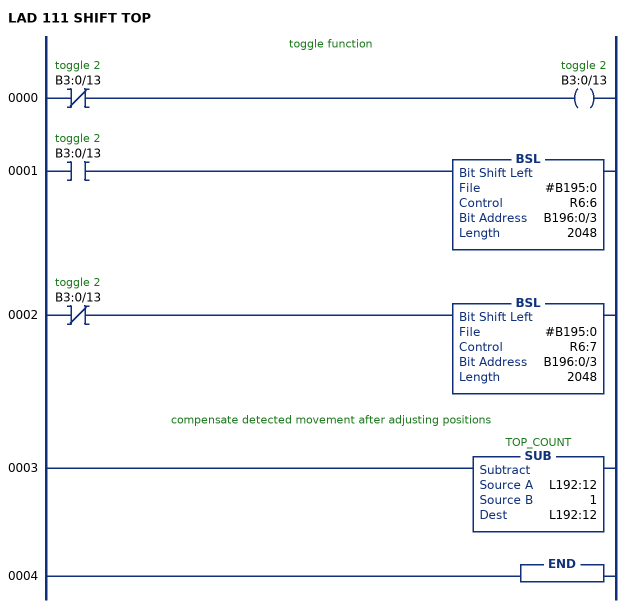
% Rung: 0 %
% toggle function %
SOR XIO B3:0/13 OTE B3:0/13 EOR
%   B3:0/13  "toggle 2" %
% Rung: 1 %
SOR XIC B3:0/13 BSL #B195:0 R6:6 B196:0/3 2048 EOR
%   B3:0/13  "toggle 2" %
%   B196:0/3  OFF %
% Rung: 2 %
SOR XIO B3:0/13 BSL #B195:0 R6:7 B196:0/3 2048 EOR
%   B3:0/13  "toggle 2" %
%   B196:0/3  OFF %
% Rung: 3 %
% compensate detected movement after adjusting positions %
SOR SUB L192:12 1 L192:12 EOR
%   L192:12  TOP_COUNT %
% Rung: 4 %
SOR END EOR

LADDER 121 "OPTIC BOT"
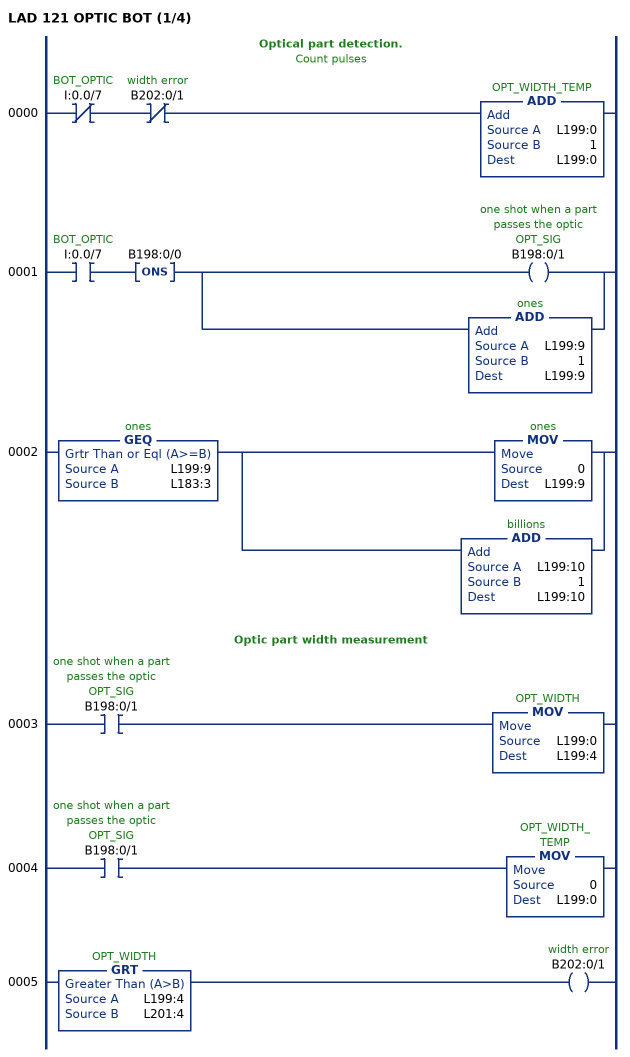
% Rung: 0 %
% TITLE: Optical part detection. %
% Count pulses %
SOR XIO I:0.0/7 XIO B202:0/1 ADD L199:0 1 L199:0 EOR
%   I:0.0/7  BOT_OPTIC %
%   B202:0/1  "width error" %
%   L199:0  OPT_WIDTH_TEMP %
% Rung: 1 %
SOR XIC I:0.0/7 ONS B198:0/0 BST OTE B198:0/1 NXB ADD L199:9 1 L199:9 BND EOR
%   I:0.0/7  BOT_OPTIC %
%   B198:0/1  OPT_SIG  "one shot when a part passes the optic" %
%   L199:9  "ones" %
% Rung: 2 %
SOR GEQ L199:9 L183:3 BST MOV 0 L199:9 NXB ADD L199:10 1 L199:10 BND EOR
%   L199:9  "ones" %
%   L183:3  "button state" %
%   L199:10  "billions" %
% Rung: 3 %
% TITLE: Optic part width measurement %
SOR XIC B198:0/1 MOV L199:0 L199:4 EOR
%   B198:0/1  OPT_SIG  "one shot when a part passes the optic" %
%   L199:0  OPT_WIDTH_TEMP %
%   L199:4  OPT_WIDTH %
% Rung: 4 %
SOR XIC B198:0/1 MOV 0 L199:0 EOR
%   B198:0/1  OPT_SIG  "one shot when a part passes the optic" %
%   L199:0  OPT_WIDTH_TEMP %
% Rung: 5 %
SOR GRT L199:4 L201:4 OTE B202:0/1 EOR
%   L199:4  OPT_WIDTH %
%   L201:4  MAX_WIDTH  "hmi in" %
%   B202:0/1  "width error" %

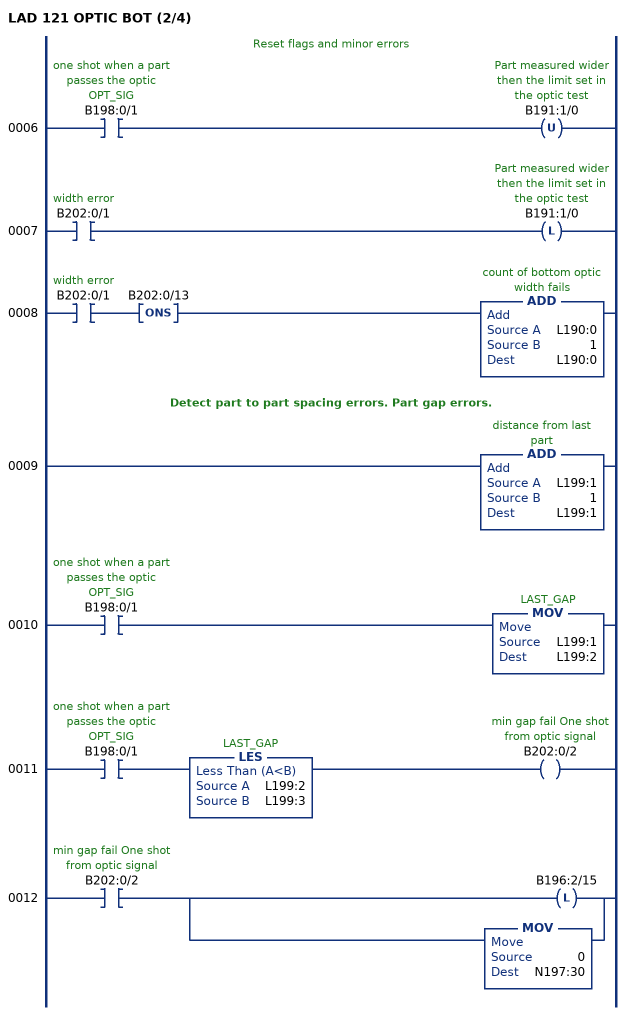
% Rung: 6 %
% Reset flags and minor errors %
SOR XIC B198:0/1 OTU B191:1/0 EOR
%   B198:0/1  OPT_SIG  "one shot when a part passes the optic" %
%   B191:1/0  "Part measured wider then the limit set in the optic test" %
% Rung: 7 %
SOR XIC B202:0/1 OTL B191:1/0 EOR
%   B202:0/1  "width error" %
%   B191:1/0  "Part measured wider then the limit set in the optic test" %
% Rung: 8 %
SOR XIC B202:0/1 ONS B202:0/13 ADD L190:0 1 L190:0 EOR
%   B202:0/1  "width error" %
%   L190:0  "count of bottom optic width fails" %
% Rung: 9 %
% TITLE: Detect part to part spacing errors. Part gap errors. %
SOR ADD L199:1 1 L199:1 EOR
%   L199:1  "distance from last part" %
% Rung: 10 %
SOR XIC B198:0/1 MOV L199:1 L199:2 EOR
%   B198:0/1  OPT_SIG  "one shot when a part passes the optic" %
%   L199:1  "distance from last part" %
%   L199:2  LAST_GAP %
% Rung: 11 %
SOR XIC B198:0/1 LES L199:2 L199:3 OTE B202:0/2 EOR
%   B198:0/1  OPT_SIG  "one shot when a part passes the optic" %
%   L199:2  LAST_GAP %
%   L199:3  MIN_WIDTH %
%   B202:0/2  "min gap fail One shot from optic signal" %
% Rung: 12 %
SOR XIC B202:0/2 BST OTL B196:2/15 NXB MOV 0 N197:30 BND EOR
%   B202:0/2  "min gap fail One shot from optic signal" %

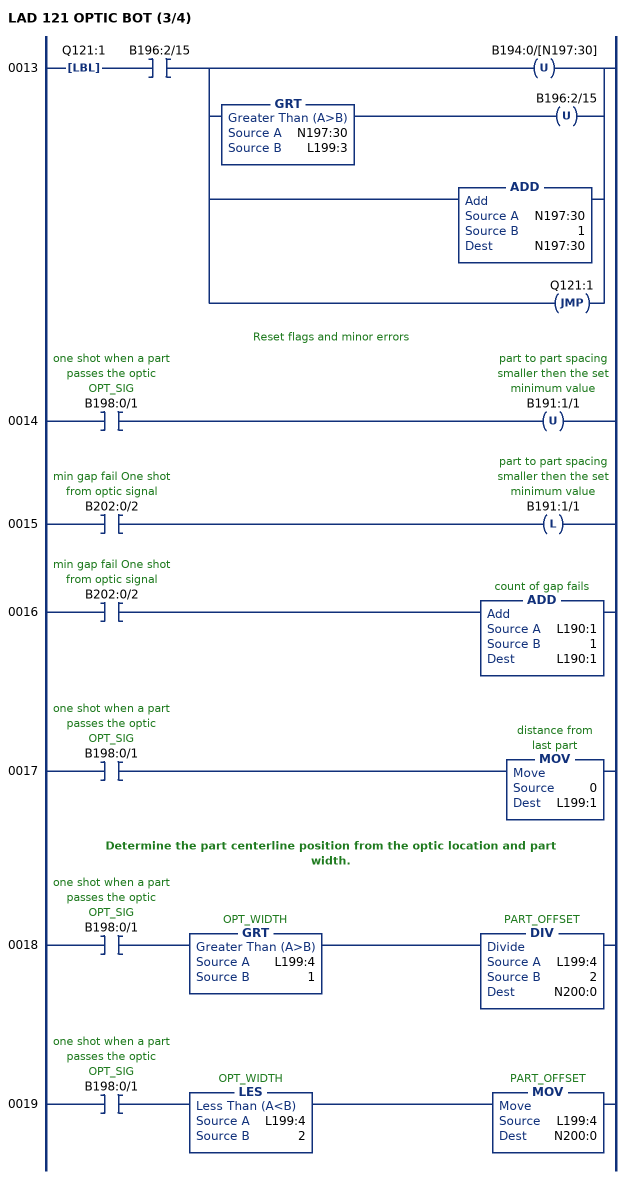
% Rung: 13 %
SOR LBL Q121:1 XIC B196:2/15 BST OTU B194:0/[N197:30] NXB GRT N197:30 L199:3 OTU B196:2/15 NXB ADD N197:30 1 N197:30 NXB JMP Q121:1 BND EOR
%   L199:3  MIN_WIDTH %
% Rung: 14 %
% Reset flags and minor errors %
SOR XIC B198:0/1 OTU B191:1/1 EOR
%   B198:0/1  OPT_SIG  "one shot when a part passes the optic" %
%   B191:1/1  "part to part spacing smaller then the set minimum value" %
% Rung: 15 %
SOR XIC B202:0/2 OTL B191:1/1 EOR
%   B202:0/2  "min gap fail One shot from optic signal" %
%   B191:1/1  "part to part spacing smaller then the set minimum value" %
% Rung: 16 %
SOR XIC B202:0/2 ADD L190:1 1 L190:1 EOR
%   B202:0/2  "min gap fail One shot from optic signal" %
%   L190:1  "count of gap fails" %
% Rung: 17 %
SOR XIC B198:0/1 MOV 0 L199:1 EOR
%   B198:0/1  OPT_SIG  "one shot when a part passes the optic" %
%   L199:1  "distance from last part" %
% Rung: 18 %
% TITLE: Determine the part centerline position from the optic location and part width. %
SOR XIC B198:0/1 GRT L199:4 1 DIV L199:4 2 N200:0 EOR
%   B198:0/1  OPT_SIG  "one shot when a part passes the optic" %
%   L199:4  OPT_WIDTH %
%   N200:0  PART_OFFSET %
% Rung: 19 %
SOR XIC B198:0/1 LES L199:4 2 MOV L199:4 N200:0 EOR
%   B198:0/1  OPT_SIG  "one shot when a part passes the optic" %
%   L199:4  OPT_WIDTH %
%   N200:0  PART_OFFSET %

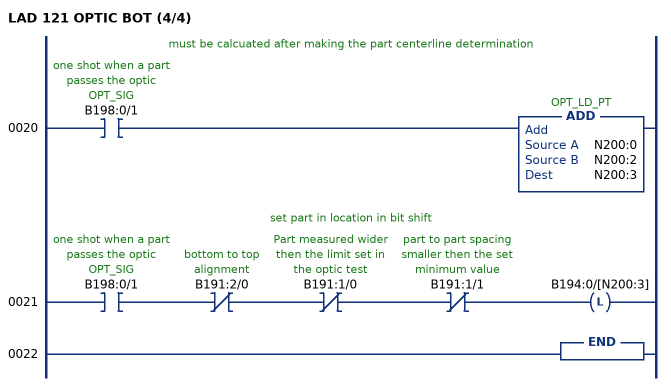
% Rung: 20 %
% must be calcuated after making the part centerline determination %
SOR XIC B198:0/1 ADD N200:0 N200:2 N200:3 EOR
%   B198:0/1  OPT_SIG  "one shot when a part passes the optic" %
%   N200:0  PART_OFFSET %
%   N200:2  OPTIC_LOC %
%   N200:3  OPT_LD_PT %
% Rung: 21 %
% set part in location in bit shift %
SOR XIC B198:0/1 XIO B191:2/0 XIO B191:1/0 XIO B191:1/1 OTL B194:0/[N200:3] EOR
%   B198:0/1  OPT_SIG  "one shot when a part passes the optic" %
%   B191:2/0  "bottom to top alignment" %
%   B191:1/0  "Part measured wider then the limit set in the optic test" %
%   B191:1/1  "part to part spacing smaller then the set minimum value" %
%   N200:3  OPT_LD_PT %
% Rung: 22 %
SOR END EOR

LADDER 125 "INS 1"
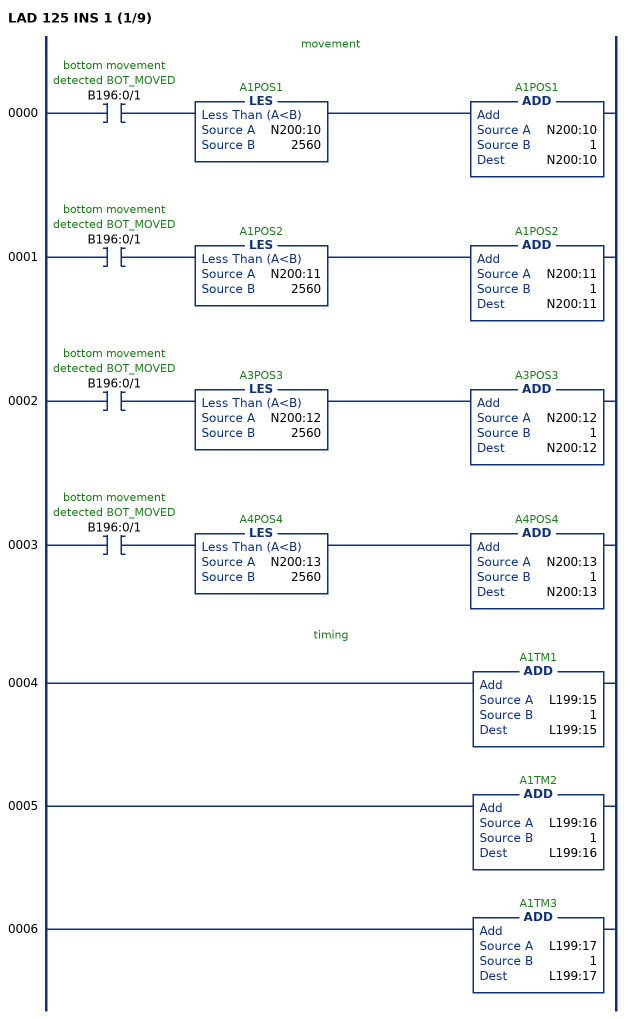
% Rung: 0 %
% movement %
SOR XIC B196:0/1 LES N200:10 2560 ADD N200:10 1 N200:10 EOR
%   B196:0/1  BOT_MOVED  "bottom movement detected" %
%   N200:10  A1POS1 %
% Rung: 1 %
SOR XIC B196:0/1 LES N200:11 2560 ADD N200:11 1 N200:11 EOR
%   B196:0/1  BOT_MOVED  "bottom movement detected" %
%   N200:11  A1POS2 %
% Rung: 2 %
SOR XIC B196:0/1 LES N200:12 2560 ADD N200:12 1 N200:12 EOR
%   B196:0/1  BOT_MOVED  "bottom movement detected" %
%   N200:12  A3POS3 %
% Rung: 3 %
SOR XIC B196:0/1 LES N200:13 2560 ADD N200:13 1 N200:13 EOR
%   B196:0/1  BOT_MOVED  "bottom movement detected" %
%   N200:13  A4POS4 %
% Rung: 4 %
% timing %
SOR ADD L199:15 1 L199:15 EOR
%   L199:15  A1TM1 %
% Rung: 5 %
SOR ADD L199:16 1 L199:16 EOR
%   L199:16  A1TM2 %
% Rung: 6 %
SOR ADD L199:17 1 L199:17 EOR
%   L199:17  A1TM3 %

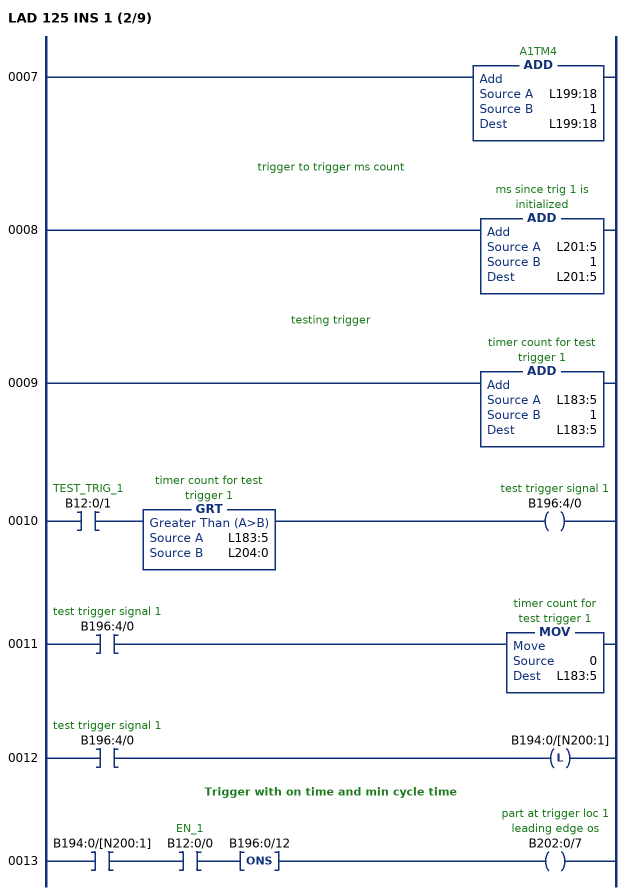
% Rung: 7 %
SOR ADD L199:18 1 L199:18 EOR
%   L199:18  A1TM4 %
% Rung: 8 %
% trigger to trigger ms count %
SOR ADD L201:5 1 L201:5 EOR
%   L201:5  "ms since trig 1 is initialized" %
% Rung: 9 %
% testing trigger %
SOR ADD L183:5 1 L183:5 EOR
%   L183:5  "timer count for test trigger 1" %
% Rung: 10 %
SOR XIC B12:0/1 GRT L183:5 L204:0 OTE B196:4/0 EOR
%   B12:0/1  TEST_TRIG_1 %
%   L183:5  "timer count for test trigger 1" %
%   B196:4/0  "test trigger signal 1" %
% Rung: 11 %
SOR XIC B196:4/0 MOV 0 L183:5 EOR
%   B196:4/0  "test trigger signal 1" %
%   L183:5  "timer count for test trigger 1" %
% Rung: 12 %
SOR XIC B196:4/0 OTL B194:0/[N200:1] EOR
%   B196:4/0  "test trigger signal 1" %
%   N200:1  INS_1_TRIG_LOC %
% Rung: 13 %
% TITLE: Trigger with on time and min cycle time %
SOR XIC B194:0/[N200:1] XIC B12:0/0 ONS B196:0/12 OTE B202:0/7 EOR
%   N200:1  INS_1_TRIG_LOC %
%   B12:0/0  EN_1 %
%   B202:0/7  "part at trigger loc 1 leading edge os" %

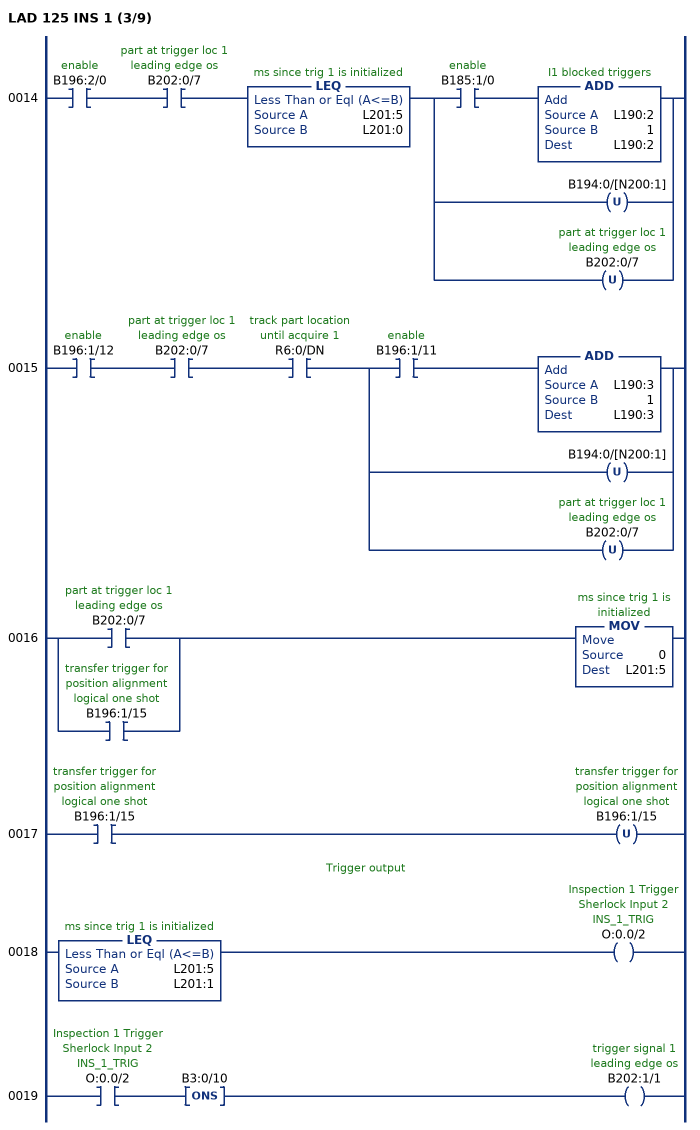
% Rung: 14 %
SOR XIC B196:2/0 XIC B202:0/7 LEQ L201:5 L201:0 BST XIC B185:1/0 ADD L190:2 1 L190:2 NXB OTU B194:0/[N200:1] NXB OTU B202:0/7 BND EOR
%   B196:2/0  "enable" %
%   B202:0/7  "part at trigger loc 1 leading edge os" %
%   L201:5  "ms since trig 1 is initialized" %
%   L201:0  CAM_1_MIN_CYCLE_TIME %
%   B185:1/0  "enable" %
%   L190:2  "I1 blocked triggers" %
%   N200:1  INS_1_TRIG_LOC %
% Rung: 15 %
SOR XIC B196:1/12 XIC B202:0/7 XIC R6:0/DN BST XIC B196:1/11 ADD L190:3 1 L190:3 NXB OTU B194:0/[N200:1] NXB OTU B202:0/7 BND EOR
%   B196:1/12  "enable" %
%   B202:0/7  "part at trigger loc 1 leading edge os" %
%   R6:0  "track part location until acquire 1" %
%   B196:1/11  "enable" %
%   N200:1  INS_1_TRIG_LOC %
% Rung: 16 %
SOR BST XIC B202:0/7 NXB XIC B196:1/15 BND MOV 0 L201:5 EOR
%   B202:0/7  "part at trigger loc 1 leading edge os" %
%   B196:1/15  "transfer trigger for position alignment logical one shot" %
%   L201:5  "ms since trig 1 is initialized" %
% Rung: 17 %
SOR XIC B196:1/15 OTU B196:1/15 EOR
%   B196:1/15  "transfer trigger for position alignment logical one shot" %
% Rung: 18 %
% Trigger output %
SOR LEQ L201:5 L201:1 OTE O:0.0/2 EOR
%   L201:5  "ms since trig 1 is initialized" %
%   L201:1  CAM_1_TRIG_TIME  "out time" %
%   O:0.0/2  INS_1_TRIG  "Inspection 1 Trigger Sherlock Input 2" %
% Rung: 19 %
SOR XIC O:0.0/2 ONS B3:0/10 OTE B202:1/1 EOR
%   O:0.0/2  INS_1_TRIG  "Inspection 1 Trigger Sherlock Input 2" %
%   B202:1/1  "trigger signal 1 leading edge os" %

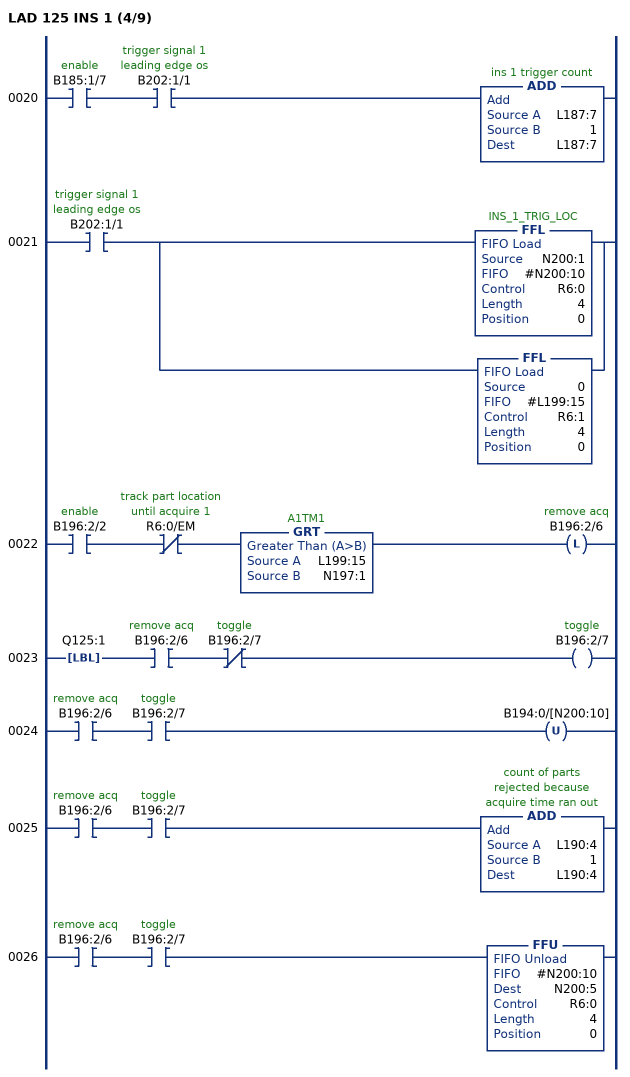
% Rung: 20 %
SOR XIC B185:1/7 XIC B202:1/1 ADD L187:7 1 L187:7 EOR
%   B185:1/7  "enable" %
%   B202:1/1  "trigger signal 1 leading edge os" %
%   L187:7  "ins 1 trigger count" %
% Rung: 21 %
SOR XIC B202:1/1 BST FFL N200:1 #N200:10 R6:0 4 0 NXB FFL 0 #L199:15 R6:1 4 0 BND EOR
%   B202:1/1  "trigger signal 1 leading edge os" %
%   N200:1  INS_1_TRIG_LOC %
%   N200:10  A1POS1 %
%   R6:0  "track part location until acquire 1" %
%   L199:15  A1TM1 %
%   R6:1  "track acquire time 1" %
% Rung: 22 %
SOR XIC B196:2/2 XIO R6:0/EM GRT L199:15 N197:1 OTL B196:2/6 EOR
%   B196:2/2  "enable" %
%   R6:0  "track part location until acquire 1" %
%   L199:15  A1TM1 %
%   N197:1  "maximim acquire time 1" %
%   B196:2/6  "remove acq" %
% Rung: 23 %
SOR LBL Q125:1 XIC B196:2/6 XIO B196:2/7 OTE B196:2/7 EOR
%   B196:2/6  "remove acq" %
%   B196:2/7  "toggle" %
% Rung: 24 %
SOR XIC B196:2/6 XIC B196:2/7 OTU B194:0/[N200:10] EOR
%   B196:2/6  "remove acq" %
%   B196:2/7  "toggle" %
%   N200:10  A1POS1 %
% Rung: 25 %
SOR XIC B196:2/6 XIC B196:2/7 ADD L190:4 1 L190:4 EOR
%   B196:2/6  "remove acq" %
%   B196:2/7  "toggle" %
%   L190:4  "count of parts rejected because acquire time ran out" %
% Rung: 26 %
SOR XIC B196:2/6 XIC B196:2/7 FFU #N200:10 N200:5 R6:0 4 0 EOR
%   B196:2/6  "remove acq" %
%   B196:2/7  "toggle" %
%   N200:10  A1POS1 %
%   R6:0  "track part location until acquire 1" %

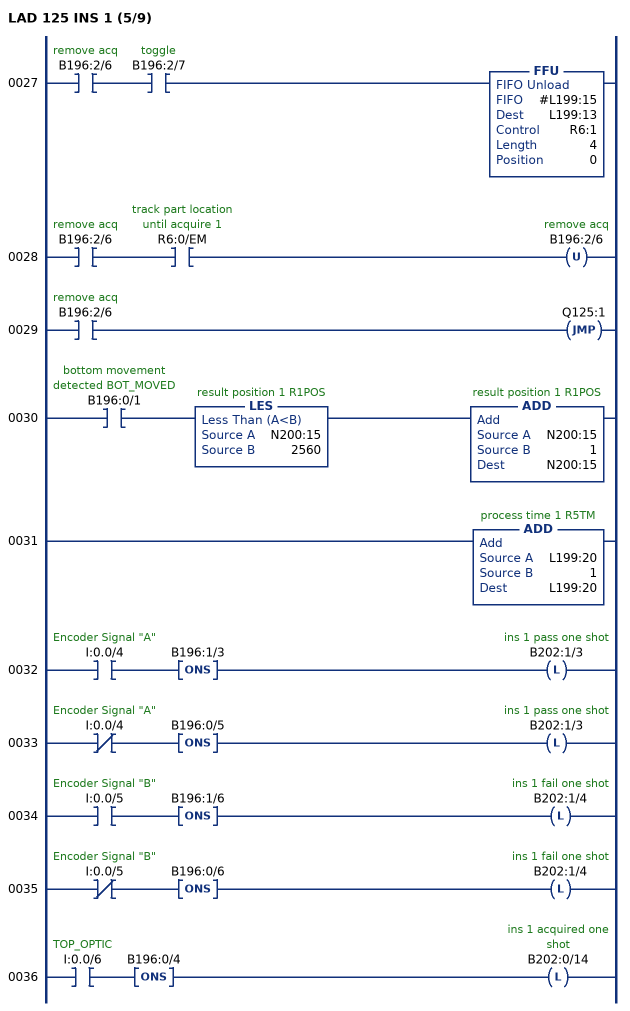
% Rung: 27 %
SOR XIC B196:2/6 XIC B196:2/7 FFU #L199:15 L199:13 R6:1 4 0 EOR
%   B196:2/6  "remove acq" %
%   B196:2/7  "toggle" %
%   L199:15  A1TM1 %
%   R6:1  "track acquire time 1" %
% Rung: 28 %
SOR XIC B196:2/6 XIC R6:0/EM OTU B196:2/6 EOR
%   B196:2/6  "remove acq" %
%   R6:0  "track part location until acquire 1" %
% Rung: 29 %
SOR XIC B196:2/6 JMP Q125:1 EOR
%   B196:2/6  "remove acq" %
% Rung: 30 %
SOR XIC B196:0/1 LES N200:15 2560 ADD N200:15 1 N200:15 EOR
%   B196:0/1  BOT_MOVED  "bottom movement detected" %
%   N200:15  R1POS  "result position 1" %
% Rung: 31 %
SOR ADD L199:20 1 L199:20 EOR
%   L199:20  R5TM  "process time 1" %
% Rung: 32 %
SOR XIC I:0.0/4 ONS B196:1/3 OTL B202:1/3 EOR
%   I:0.0/4  "Encoder Signal "A"" %
%   B202:1/3  "ins 1 pass one shot" %
% Rung: 33 %
SOR XIO I:0.0/4 ONS B196:0/5 OTL B202:1/3 EOR
%   I:0.0/4  "Encoder Signal "A"" %
%   B202:1/3  "ins 1 pass one shot" %
% Rung: 34 %
SOR XIC I:0.0/5 ONS B196:1/6 OTL B202:1/4 EOR
%   I:0.0/5  "Encoder Signal "B"" %
%   B202:1/4  "ins 1 fail one shot" %
% Rung: 35 %
SOR XIO I:0.0/5 ONS B196:0/6 OTL B202:1/4 EOR
%   I:0.0/5  "Encoder Signal "B"" %
%   B202:1/4  "ins 1 fail one shot" %
% Rung: 36 %
SOR XIC I:0.0/6 ONS B196:0/4 OTL B202:0/14 EOR
%   I:0.0/6  TOP_OPTIC %
%   B202:0/14  "ins 1 acquired one shot" %

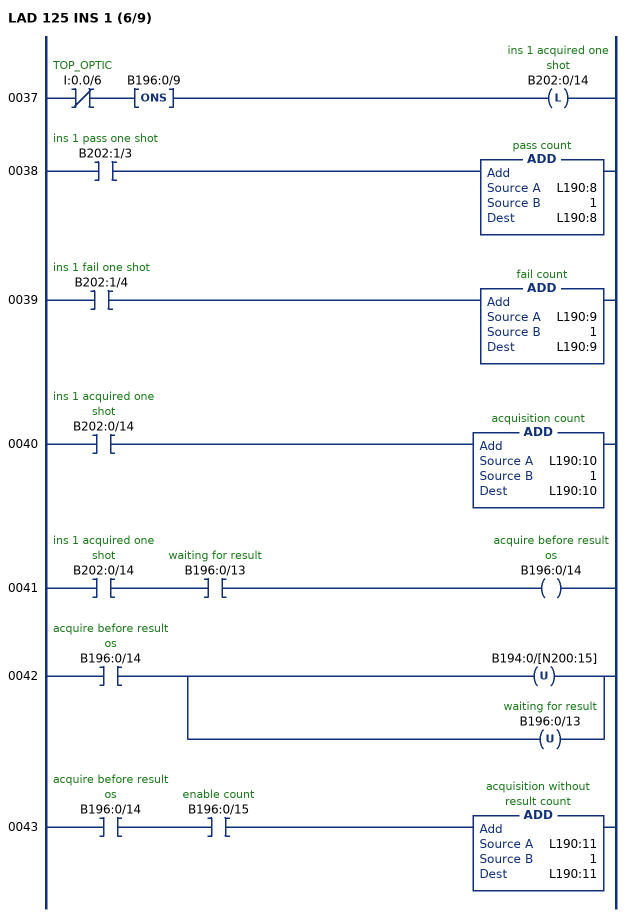
% Rung: 37 %
SOR XIO I:0.0/6 ONS B196:0/9 OTL B202:0/14 EOR
%   I:0.0/6  TOP_OPTIC %
%   B202:0/14  "ins 1 acquired one shot" %
% Rung: 38 %
SOR XIC B202:1/3 ADD L190:8 1 L190:8 EOR
%   B202:1/3  "ins 1 pass one shot" %
%   L190:8  "pass count" %
% Rung: 39 %
SOR XIC B202:1/4 ADD L190:9 1 L190:9 EOR
%   B202:1/4  "ins 1 fail one shot" %
%   L190:9  "fail count" %
% Rung: 40 %
SOR XIC B202:0/14 ADD L190:10 1 L190:10 EOR
%   B202:0/14  "ins 1 acquired one shot" %
%   L190:10  "acquisition count" %
% Rung: 41 %
SOR XIC B202:0/14 XIC B196:0/13 OTE B196:0/14 EOR
%   B202:0/14  "ins 1 acquired one shot" %
%   B196:0/13  "waiting for result" %
%   B196:0/14  "acquire before result os" %
% Rung: 42 %
SOR XIC B196:0/14 BST OTU B194:0/[N200:15] NXB OTU B196:0/13 BND EOR
%   B196:0/14  "acquire before result os" %
%   N200:15  R1POS  "result position 1" %
%   B196:0/13  "waiting for result" %
% Rung: 43 %
SOR XIC B196:0/14 XIC B196:0/15 ADD L190:11 1 L190:11 EOR
%   B196:0/14  "acquire before result os" %
%   B196:0/15  "enable count" %
%   L190:11  "acquisition without result count" %

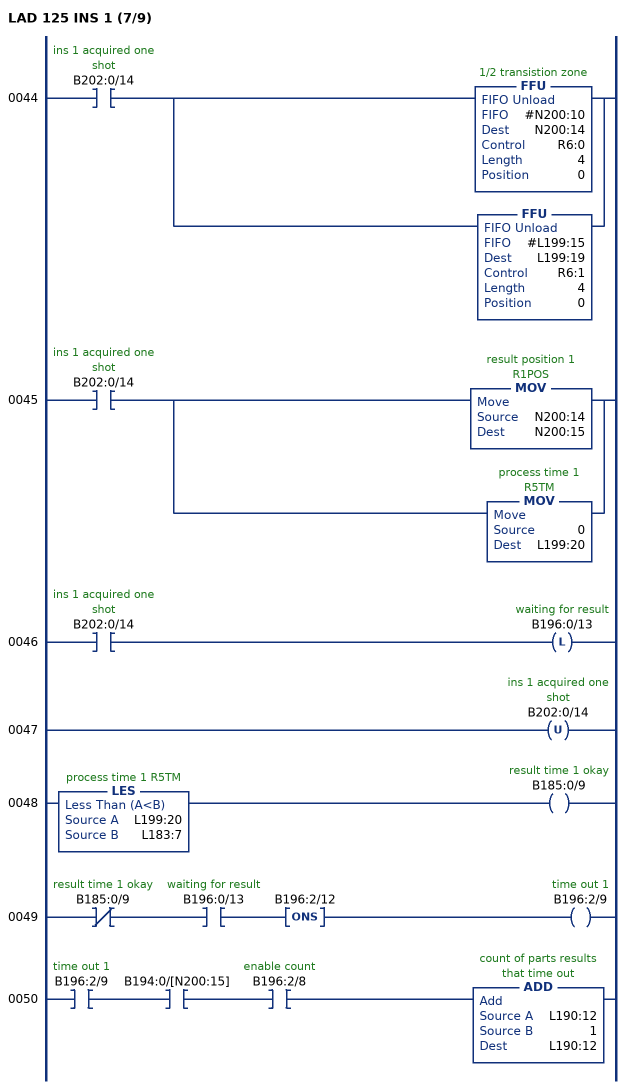
% Rung: 44 %
SOR XIC B202:0/14 BST FFU #N200:10 N200:14 R6:0 4 0 NXB FFU #L199:15 L199:19 R6:1 4 0 BND EOR
%   B202:0/14  "ins 1 acquired one shot" %
%   N200:10  A1POS1 %
%   N200:14  "1/2 transistion zone" %
%   R6:0  "track part location until acquire 1" %
%   L199:15  A1TM1 %
%   R6:1  "track acquire time 1" %
% Rung: 45 %
SOR XIC B202:0/14 BST MOV N200:14 N200:15 NXB MOV 0 L199:20 BND EOR
%   B202:0/14  "ins 1 acquired one shot" %
%   N200:14  "1/2 transistion zone" %
%   N200:15  R1POS  "result position 1" %
%   L199:20  R5TM  "process time 1" %
% Rung: 46 %
SOR XIC B202:0/14 OTL B196:0/13 EOR
%   B202:0/14  "ins 1 acquired one shot" %
%   B196:0/13  "waiting for result" %
% Rung: 47 %
SOR OTU B202:0/14 EOR
%   B202:0/14  "ins 1 acquired one shot" %
% Rung: 48 %
SOR LES L199:20 L183:7 OTE B185:0/9 EOR
%   L199:20  R5TM  "process time 1" %
%   L183:7  "max process time 1" %
%   B185:0/9  "result time 1 okay" %
% Rung: 49 %
SOR XIO B185:0/9 XIC B196:0/13 ONS B196:2/12 OTE B196:2/9 EOR
%   B185:0/9  "result time 1 okay" %
%   B196:0/13  "waiting for result" %
%   B196:2/9  "time out 1" %
% Rung: 50 %
SOR XIC B196:2/9 XIC B194:0/[N200:15] XIC B196:2/8 ADD L190:12 1 L190:12 EOR
%   B196:2/9  "time out 1" %
%   N200:15  R1POS  "result position 1" %
%   B196:2/8  "enable count" %
%   L190:12  "count of parts results that time out" %

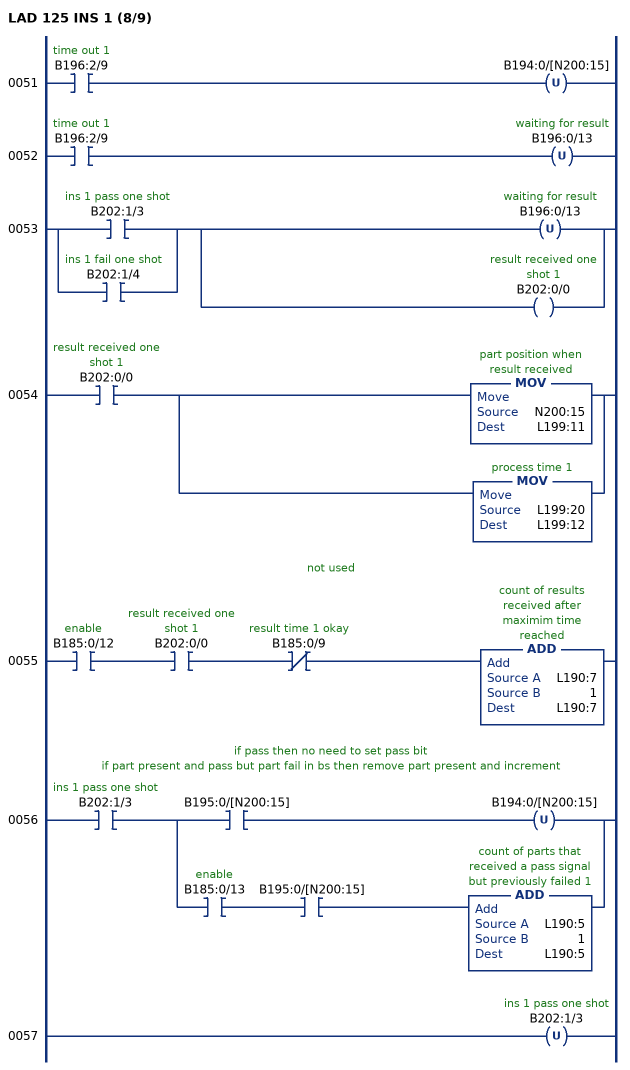
% Rung: 51 %
SOR XIC B196:2/9 OTU B194:0/[N200:15] EOR
%   B196:2/9  "time out 1" %
%   N200:15  R1POS  "result position 1" %
% Rung: 52 %
SOR XIC B196:2/9 OTU B196:0/13 EOR
%   B196:2/9  "time out 1" %
%   B196:0/13  "waiting for result" %
% Rung: 53 %
SOR BST XIC B202:1/3 NXB XIC B202:1/4 BND BST OTU B196:0/13 NXB OTE B202:0/0 BND EOR
%   B202:1/3  "ins 1 pass one shot" %
%   B202:1/4  "ins 1 fail one shot" %
%   B196:0/13  "waiting for result" %
%   B202:0/0  "result received one shot 1" %
% Rung: 54 %
SOR XIC B202:0/0 BST MOV N200:15 L199:11 NXB MOV L199:20 L199:12 BND EOR
%   B202:0/0  "result received one shot 1" %
%   N200:15  R1POS  "result position 1" %
%   L199:11  "part position when result received" %
%   L199:20  R5TM  "process time 1" %
%   L199:12  "process time 1" %
% Rung: 55 %
% not used %
SOR XIC B185:0/12 XIC B202:0/0 XIO B185:0/9 ADD L190:7 1 L190:7 EOR
%   B185:0/12  "enable" %
%   B202:0/0  "result received one shot 1" %
%   B185:0/9  "result time 1 okay" %
%   L190:7  "count of results received after maximim time reached" %
% Rung: 56 %
% if pass then no need to set pass bit
% if part present and pass but part fail in bs then remove part present and increment %
SOR XIC B202:1/3 BST XIC B195:0/[N200:15] OTU B194:0/[N200:15] NXB XIC B185:0/13 XIC B195:0/[N200:15] ADD L190:5 1 L190:5 BND EOR
%   B202:1/3  "ins 1 pass one shot" %
%   N200:15  R1POS  "result position 1" %
%   B185:0/13  "enable" %
%   L190:5  "count of parts that received a pass signal but previously failed 1" %
% Rung: 57 %
SOR OTU B202:1/3 EOR
%   B202:1/3  "ins 1 pass one shot" %

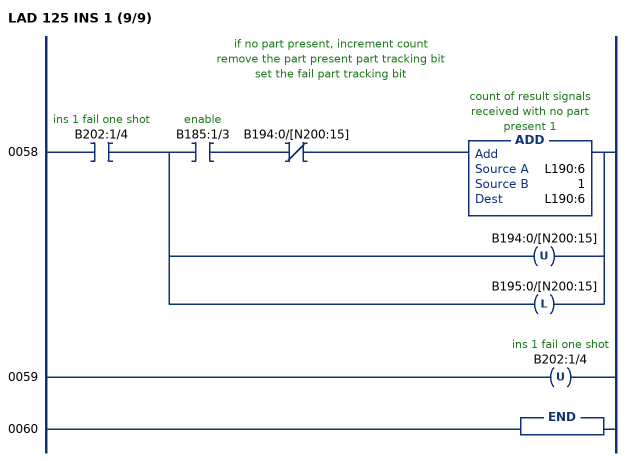
% Rung: 58 %
% if no part present, increment count
% remove the part present part tracking bit
% set the fail part tracking bit %
SOR XIC B202:1/4 BST XIC B185:1/3 XIO B194:0/[N200:15] ADD L190:6 1 L190:6 NXB OTU B194:0/[N200:15] NXB OTL B195:0/[N200:15] BND EOR
%   B202:1/4  "ins 1 fail one shot" %
%   B185:1/3  "enable" %
%   N200:15  R1POS  "result position 1" %
%   L190:6  "count of result signals received with no part present 1" %
% Rung: 59 %
SOR OTU B202:1/4 EOR
%   B202:1/4  "ins 1 fail one shot" %
% Rung: 60 %
SOR END EOR

LADDER 130 "XFER"
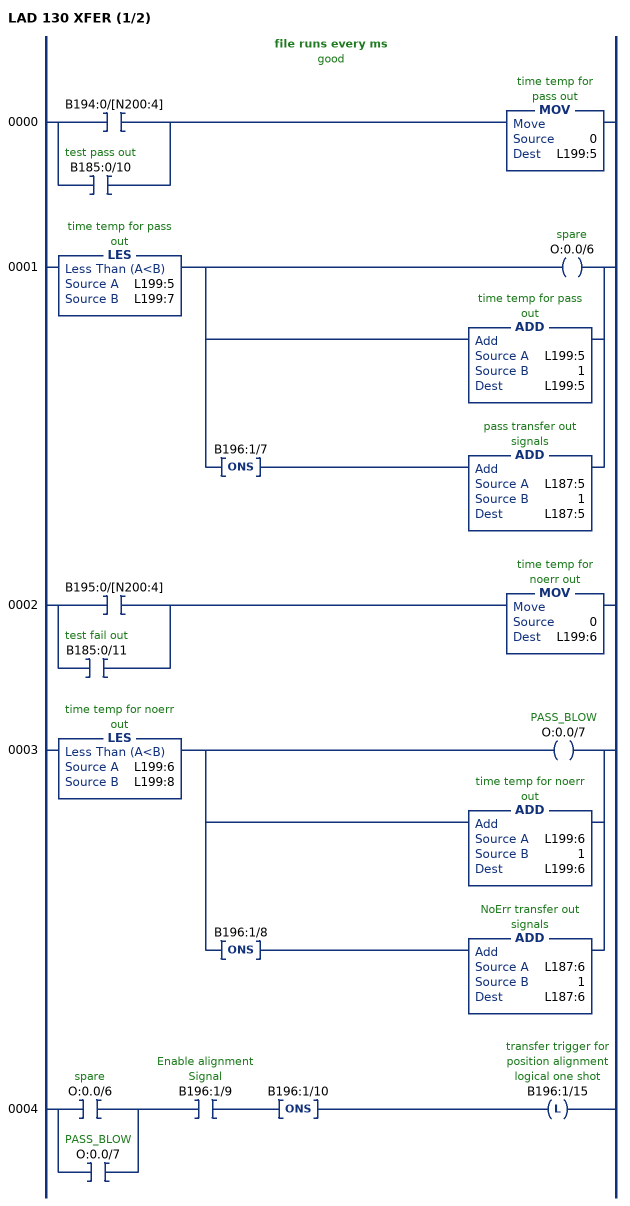
% Rung: 0 %
% TITLE: file runs every ms %
% good %
SOR BST XIC B194:0/[N200:4] NXB XIC B185:0/10 BND MOV 0 L199:5 EOR
%   N200:4  XFER_OUT  "The location to send the data out to the other inspection" %
%   B185:0/10  "test pass out" %
%   L199:5  "time temp for pass out" %
% Rung: 1 %
SOR LES L199:5 L199:7 BST OTE O:0.0/6 NXB ADD L199:5 1 L199:5 NXB ONS B196:1/7 ADD L187:5 1 L187:5 BND EOR
%   L199:5  "time temp for pass out" %
%   O:0.0/6  "spare" %
%   L187:5  "pass transfer out signals" %
% Rung: 2 %
SOR BST XIC B195:0/[N200:4] NXB XIC B185:0/11 BND MOV 0 L199:6 EOR
%   N200:4  XFER_OUT  "The location to send the data out to the other inspection" %
%   B185:0/11  "test fail out" %
%   L199:6  "time temp for noerr out" %
% Rung: 3 %
SOR LES L199:6 L199:8 BST OTE O:0.0/7 NXB ADD L199:6 1 L199:6 NXB ONS B196:1/8 ADD L187:6 1 L187:6 BND EOR
%   L199:6  "time temp for noerr out" %
%   O:0.0/7  PASS_BLOW %
%   L187:6  "NoErr transfer out signals" %
% Rung: 4 %
SOR BST XIC O:0.0/6 NXB XIC O:0.0/7 BND XIC B196:1/9 ONS B196:1/10 OTL B196:1/15 EOR
%   O:0.0/6  "spare" %
%   O:0.0/7  PASS_BLOW %
%   B196:1/9  "Enable alignment Signal" %
%   B196:1/15  "transfer trigger for position alignment logical one shot" %

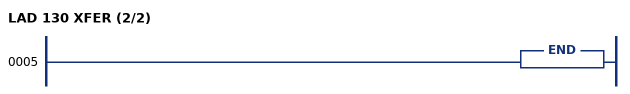
% Rung: 5 %
SOR END EOR

LADDER 140 "OPTIC TOP"
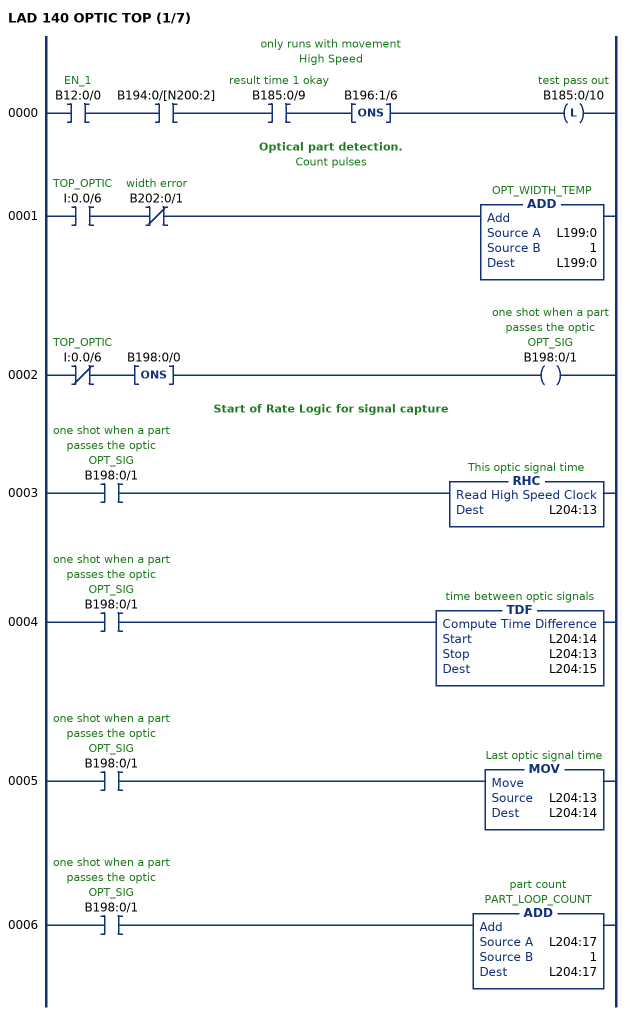
% Rung: 0 %
% only runs with movement
% High Speed %
SOR XIC B12:0/0 XIC B194:0/[N200:2] XIC B185:0/9 ONS B196:1/6 OTL B185:0/10 EOR
%   B12:0/0  EN_1 %
%   N200:2  OPTIC_LOC %
%   B185:0/9  "result time 1 okay" %
%   B185:0/10  "test pass out" %
% Rung: 1 %
% TITLE: Optical part detection. %
% Count pulses %
SOR XIC I:0.0/6 XIO B202:0/1 ADD L199:0 1 L199:0 EOR
%   I:0.0/6  TOP_OPTIC %
%   B202:0/1  "width error" %
%   L199:0  OPT_WIDTH_TEMP %
% Rung: 2 %
SOR XIO I:0.0/6 ONS B198:0/0 OTE B198:0/1 EOR
%   I:0.0/6  TOP_OPTIC %
%   B198:0/1  OPT_SIG  "one shot when a part passes the optic" %
% Rung: 3 %
% TITLE: Start of Rate Logic for signal capture %
SOR XIC B198:0/1 RHC L204:13 EOR
%   B198:0/1  OPT_SIG  "one shot when a part passes the optic" %
%   L204:13  "This optic signal time" %
% Rung: 4 %
SOR XIC B198:0/1 TDF L204:14 L204:13 L204:15 EOR
%   B198:0/1  OPT_SIG  "one shot when a part passes the optic" %
%   L204:14  "Last optic signal time" %
%   L204:13  "This optic signal time" %
%   L204:15  "time between optic signals" %
% Rung: 5 %
SOR XIC B198:0/1 MOV L204:13 L204:14 EOR
%   B198:0/1  OPT_SIG  "one shot when a part passes the optic" %
%   L204:13  "This optic signal time" %
%   L204:14  "Last optic signal time" %
% Rung: 6 %
SOR XIC B198:0/1 ADD L204:17 1 L204:17 EOR
%   B198:0/1  OPT_SIG  "one shot when a part passes the optic" %
%   L204:17  PART_LOOP_COUNT  "part count" %

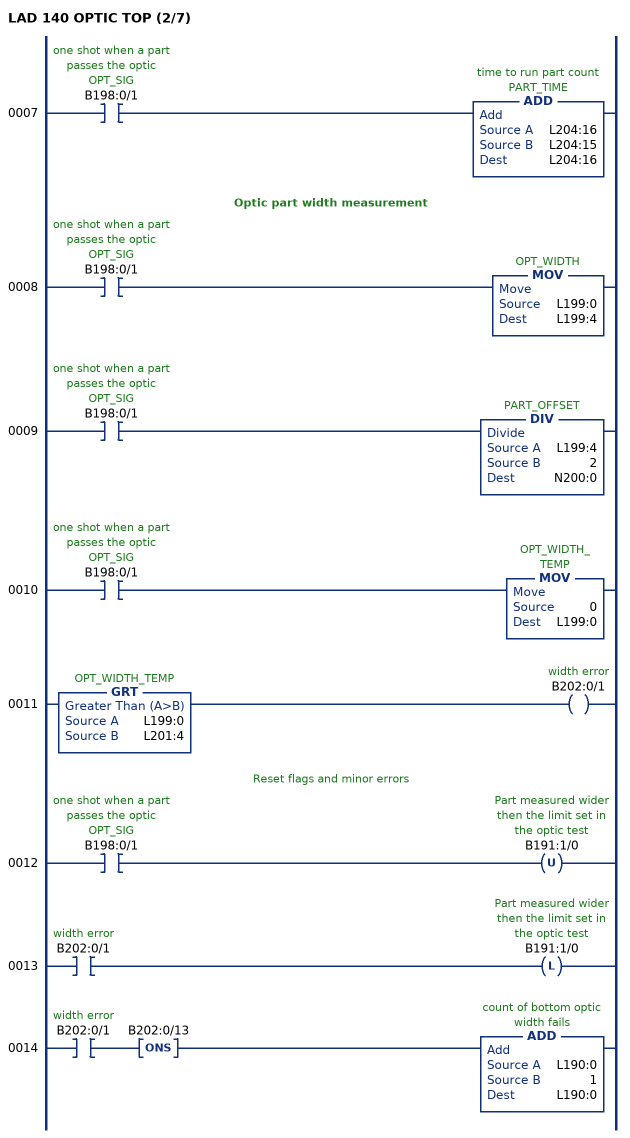
% Rung: 7 %
SOR XIC B198:0/1 ADD L204:16 L204:15 L204:16 EOR
%   B198:0/1  OPT_SIG  "one shot when a part passes the optic" %
%   L204:16  PART_TIME  "time to run part count" %
%   L204:15  "time between optic signals" %
% Rung: 8 %
% TITLE: Optic part width measurement %
SOR XIC B198:0/1 MOV L199:0 L199:4 EOR
%   B198:0/1  OPT_SIG  "one shot when a part passes the optic" %
%   L199:0  OPT_WIDTH_TEMP %
%   L199:4  OPT_WIDTH %
% Rung: 9 %
SOR XIC B198:0/1 DIV L199:4 2 N200:0 EOR
%   B198:0/1  OPT_SIG  "one shot when a part passes the optic" %
%   L199:4  OPT_WIDTH %
%   N200:0  PART_OFFSET %
% Rung: 10 %
SOR XIC B198:0/1 MOV 0 L199:0 EOR
%   B198:0/1  OPT_SIG  "one shot when a part passes the optic" %
%   L199:0  OPT_WIDTH_TEMP %
% Rung: 11 %
SOR GRT L199:0 L201:4 OTE B202:0/1 EOR
%   L199:0  OPT_WIDTH_TEMP %
%   L201:4  MAX_WIDTH  "hmi in" %
%   B202:0/1  "width error" %
% Rung: 12 %
% Reset flags and minor errors %
SOR XIC B198:0/1 OTU B191:1/0 EOR
%   B198:0/1  OPT_SIG  "one shot when a part passes the optic" %
%   B191:1/0  "Part measured wider then the limit set in the optic test" %
% Rung: 13 %
SOR XIC B202:0/1 OTL B191:1/0 EOR
%   B202:0/1  "width error" %
%   B191:1/0  "Part measured wider then the limit set in the optic test" %
% Rung: 14 %
SOR XIC B202:0/1 ONS B202:0/13 ADD L190:0 1 L190:0 EOR
%   B202:0/1  "width error" %
%   L190:0  "count of bottom optic width fails" %

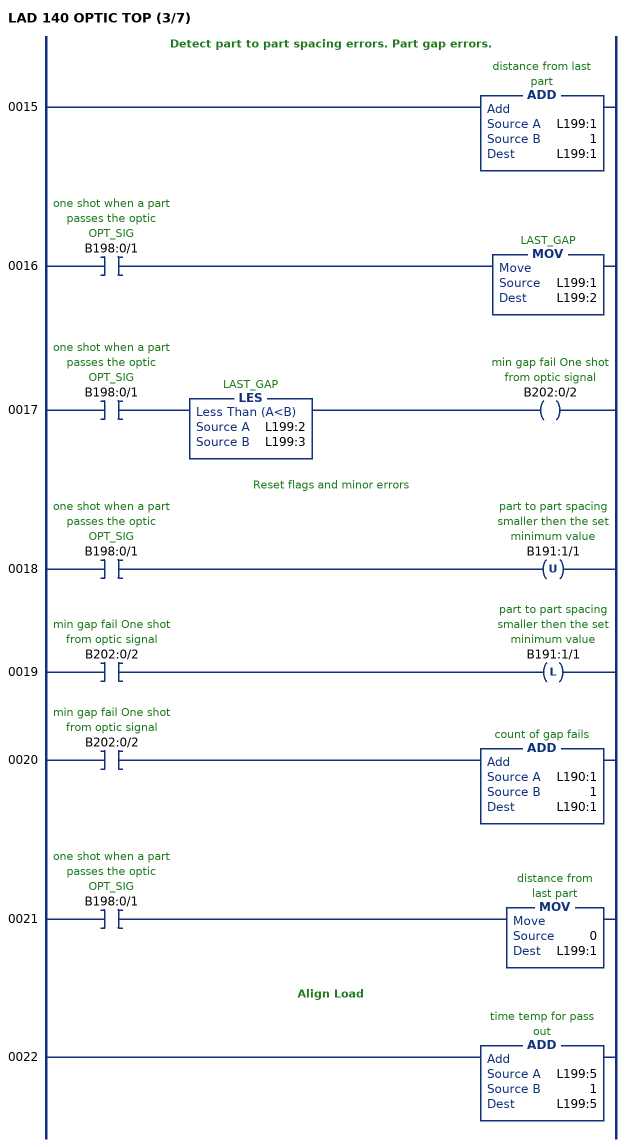
% Rung: 15 %
% TITLE: Detect part to part spacing errors. Part gap errors. %
SOR ADD L199:1 1 L199:1 EOR
%   L199:1  "distance from last part" %
% Rung: 16 %
SOR XIC B198:0/1 MOV L199:1 L199:2 EOR
%   B198:0/1  OPT_SIG  "one shot when a part passes the optic" %
%   L199:1  "distance from last part" %
%   L199:2  LAST_GAP %
% Rung: 17 %
SOR XIC B198:0/1 LES L199:2 L199:3 OTE B202:0/2 EOR
%   B198:0/1  OPT_SIG  "one shot when a part passes the optic" %
%   L199:2  LAST_GAP %
%   L199:3  MIN_WIDTH %
%   B202:0/2  "min gap fail One shot from optic signal" %
% Rung: 18 %
% Reset flags and minor errors %
SOR XIC B198:0/1 OTU B191:1/1 EOR
%   B198:0/1  OPT_SIG  "one shot when a part passes the optic" %
%   B191:1/1  "part to part spacing smaller then the set minimum value" %
% Rung: 19 %
SOR XIC B202:0/2 OTL B191:1/1 EOR
%   B202:0/2  "min gap fail One shot from optic signal" %
%   B191:1/1  "part to part spacing smaller then the set minimum value" %
% Rung: 20 %
SOR XIC B202:0/2 ADD L190:1 1 L190:1 EOR
%   B202:0/2  "min gap fail One shot from optic signal" %
%   L190:1  "count of gap fails" %
% Rung: 21 %
SOR XIC B198:0/1 MOV 0 L199:1 EOR
%   B198:0/1  OPT_SIG  "one shot when a part passes the optic" %
%   L199:1  "distance from last part" %
% Rung: 22 %
% TITLE: Align Load %
SOR ADD L199:5 1 L199:5 EOR
%   L199:5  "time temp for pass out" %

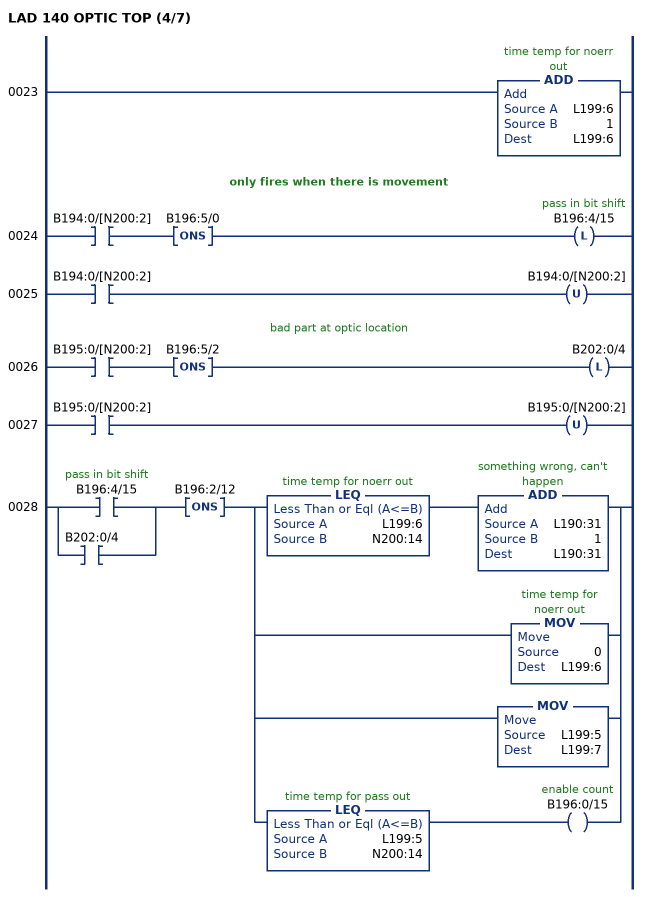
% Rung: 23 %
SOR ADD L199:6 1 L199:6 EOR
%   L199:6  "time temp for noerr out" %
% Rung: 24 %
% TITLE: only fires when there is movement %
SOR XIC B194:0/[N200:2] ONS B196:5/0 OTL B196:4/15 EOR
%   N200:2  OPTIC_LOC %
%   B196:4/15  "pass in bit shift" %
% Rung: 25 %
SOR XIC B194:0/[N200:2] OTU B194:0/[N200:2] EOR
%   N200:2  OPTIC_LOC %
% Rung: 26 %
% bad part at optic location %
SOR XIC B195:0/[N200:2] ONS B196:5/2 OTL B202:0/4 EOR
%   N200:2  OPTIC_LOC %
% Rung: 27 %
SOR XIC B195:0/[N200:2] OTU B195:0/[N200:2] EOR
%   N200:2  OPTIC_LOC %
% Rung: 28 %
SOR BST XIC B196:4/15 NXB XIC B202:0/4 BND ONS B196:2/12 BST LEQ L199:6 N200:14 ADD L190:31 1 L190:31 NXB MOV 0 L199:6 NXB MOV L199:5 L199:7 NXB LEQ L199:5 N200:14 OTE B196:0/15 BND EOR
%   B196:4/15  "pass in bit shift" %
%   L199:6  "time temp for noerr out" %
%   N200:14  "1/2 transistion zone" %
%   L190:31  "something wrong, can't happen" %
%   L199:5  "time temp for pass out" %
%   B196:0/15  "enable count" %

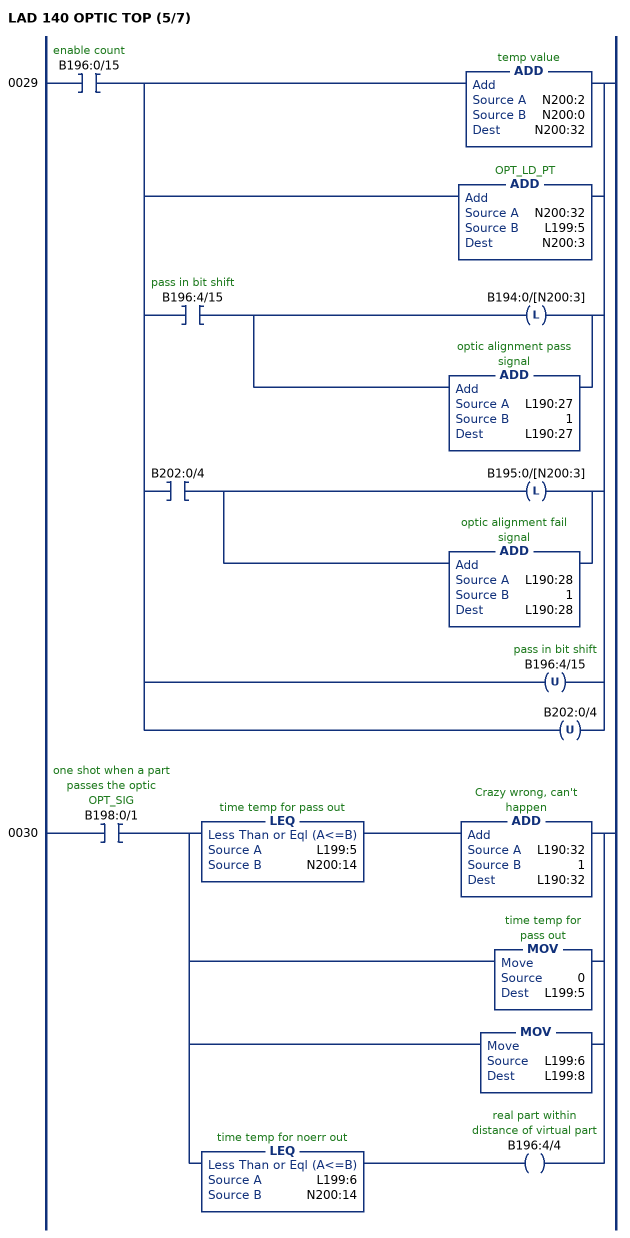
% Rung: 29 %
SOR XIC B196:0/15 BST ADD N200:2 N200:0 N200:32 NXB ADD N200:32 L199:5 N200:3 NXB XIC B196:4/15 BST OTL B194:0/[N200:3] NXB ADD L190:27 1 L190:27 BND NXB XIC B202:0/4 BST OTL B195:0/[N200:3] NXB ADD L190:28 1 L190:28 BND NXB OTU B196:4/15 NXB OTU B202:0/4 BND EOR
%   B196:0/15  "enable count" %
%   N200:2  OPTIC_LOC %
%   N200:0  PART_OFFSET %
%   N200:32  "temp value" %
%   L199:5  "time temp for pass out" %
%   N200:3  OPT_LD_PT %
%   B196:4/15  "pass in bit shift" %
%   L190:27  "optic alignment pass signal" %
%   L190:28  "optic alignment fail signal" %
% Rung: 30 %
SOR XIC B198:0/1 BST LEQ L199:5 N200:14 ADD L190:32 1 L190:32 NXB MOV 0 L199:5 NXB MOV L199:6 L199:8 NXB LEQ L199:6 N200:14 OTE B196:4/4 BND EOR
%   B198:0/1  OPT_SIG  "one shot when a part passes the optic" %
%   L199:5  "time temp for pass out" %
%   N200:14  "1/2 transistion zone" %
%   L190:32  "Crazy wrong, can't happen" %
%   L199:6  "time temp for noerr out" %
%   B196:4/4  "real part within distance of virtual part" %

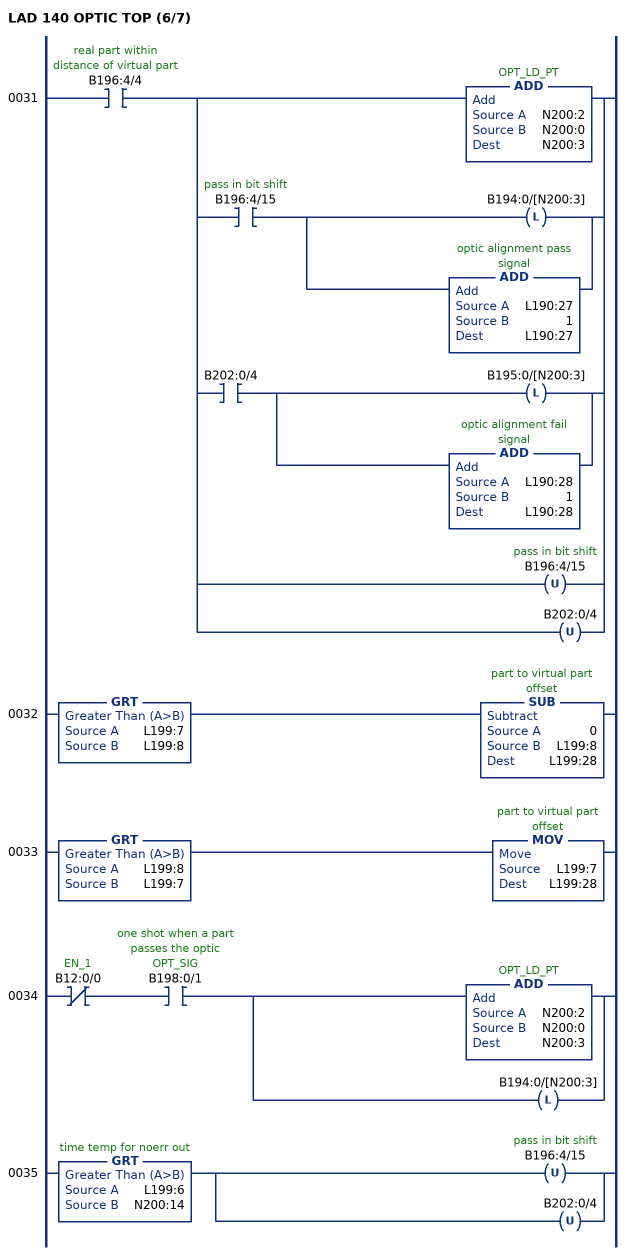
% Rung: 31 %
SOR XIC B196:4/4 BST ADD N200:2 N200:0 N200:3 NXB XIC B196:4/15 BST OTL B194:0/[N200:3] NXB ADD L190:27 1 L190:27 BND NXB XIC B202:0/4 BST OTL B195:0/[N200:3] NXB ADD L190:28 1 L190:28 BND NXB OTU B196:4/15 NXB OTU B202:0/4 BND EOR
%   B196:4/4  "real part within distance of virtual part" %
%   N200:2  OPTIC_LOC %
%   N200:0  PART_OFFSET %
%   N200:3  OPT_LD_PT %
%   B196:4/15  "pass in bit shift" %
%   L190:27  "optic alignment pass signal" %
%   L190:28  "optic alignment fail signal" %
% Rung: 32 %
SOR GRT L199:7 L199:8 SUB 0 L199:8 L199:28 EOR
%   L199:28  "part to virtual part offset" %
% Rung: 33 %
SOR GRT L199:8 L199:7 MOV L199:7 L199:28 EOR
%   L199:28  "part to virtual part offset" %
% Rung: 34 %
SOR XIO B12:0/0 XIC B198:0/1 BST ADD N200:2 N200:0 N200:3 NXB OTL B194:0/[N200:3] BND EOR
%   B12:0/0  EN_1 %
%   B198:0/1  OPT_SIG  "one shot when a part passes the optic" %
%   N200:2  OPTIC_LOC %
%   N200:0  PART_OFFSET %
%   N200:3  OPT_LD_PT %
% Rung: 35 %
SOR GRT L199:6 N200:14 BST OTU B196:4/15 NXB OTU B202:0/4 BND EOR
%   L199:6  "time temp for noerr out" %
%   N200:14  "1/2 transistion zone" %
%   B196:4/15  "pass in bit shift" %

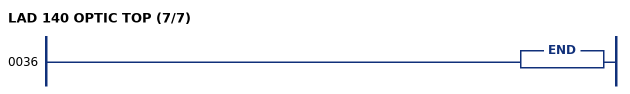
% Rung: 36 %
SOR END EOR

LADDER 150 "INS 5"
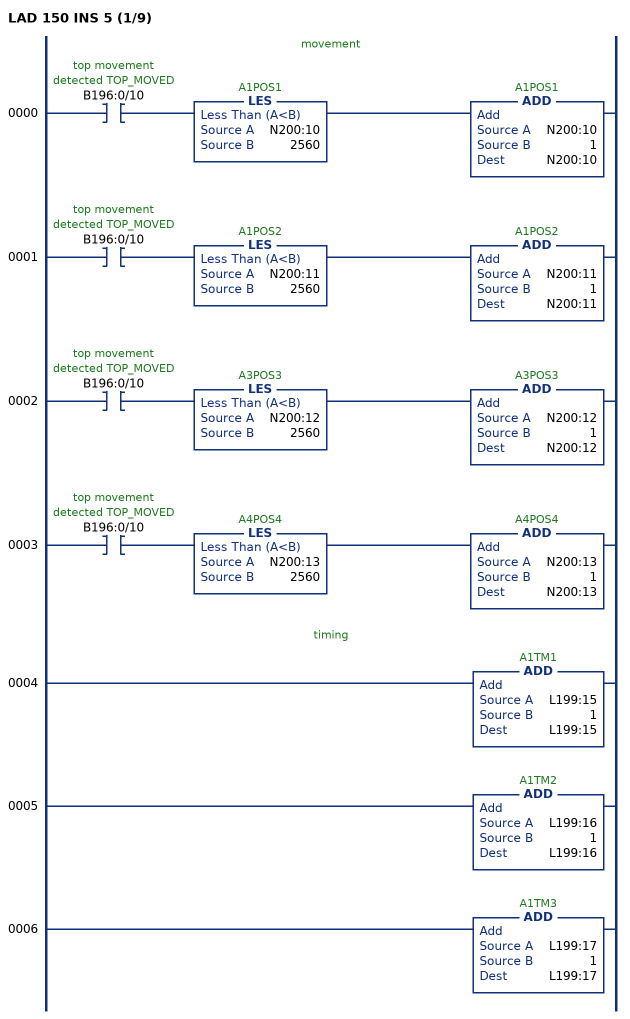
% Rung: 0 %
% movement %
SOR XIC B196:0/10 LES N200:10 2560 ADD N200:10 1 N200:10 EOR
%   B196:0/10  TOP_MOVED  "top movement detected" %
%   N200:10  A1POS1 %
% Rung: 1 %
SOR XIC B196:0/10 LES N200:11 2560 ADD N200:11 1 N200:11 EOR
%   B196:0/10  TOP_MOVED  "top movement detected" %
%   N200:11  A1POS2 %
% Rung: 2 %
SOR XIC B196:0/10 LES N200:12 2560 ADD N200:12 1 N200:12 EOR
%   B196:0/10  TOP_MOVED  "top movement detected" %
%   N200:12  A3POS3 %
% Rung: 3 %
SOR XIC B196:0/10 LES N200:13 2560 ADD N200:13 1 N200:13 EOR
%   B196:0/10  TOP_MOVED  "top movement detected" %
%   N200:13  A4POS4 %
% Rung: 4 %
% timing %
SOR ADD L199:15 1 L199:15 EOR
%   L199:15  A1TM1 %
% Rung: 5 %
SOR ADD L199:16 1 L199:16 EOR
%   L199:16  A1TM2 %
% Rung: 6 %
SOR ADD L199:17 1 L199:17 EOR
%   L199:17  A1TM3 %

